_CFC_ (* Continuous Function Chart, elements in execution order *)
#0 OR(SCHU_P2_2_UE3_T_RESET, SCHU_P2_2_SB)
#1 SEL(UE3_T_FILTER_ON, T#0ms, T#2s)
#2 fb_UE3_T:ISTOK_ANALOGVH(enable: TRUE, rawValue: SCHU_P2_2_UE3_AI1, reset: #0, enableLimitCtrl: TRUE, ctrlVoltage: NOT UE3_T_CVOLT, changeValueWithoutPower: TRUE, highRange: UE_T_HIGHRANGE, lowRange: UE_T_LOWRANGE, highLimit: SCHU_P2_2_UE_T_HIGHLIMIT, lowLimit: SCHU_P2_2_UE_T_LOWLIMIT, filterTime: #1, offset: ofset, delayEnable: TE_DELAY)
#3 SCHU_P2_2_UE3_T_VN <= #2.presentValue
#4 SCHU_P2_2_UE3_T_DOST <= #2.reliability
#5 SUB(SCHU_P2_2_UE3_T_UST, 0.6)
#6 fb_UE3_m_UST:ISTOK_LT(dost: #2.reliability, x: #2.presentValue, ust: #5, shkal: -, gist: 0.5)
#7 SCHU_P2_2_UE3_TE_M_UST <= #6.Xm
#8 SCHU_P2_2_UE3_TE_B_UST <= #6.XmN
_END_CFC_
(* the same logic as Structured Text *)
fb_UE3_T(enable := TRUE, rawValue := SCHU_P2_2_UE3_AI1, reset := SCHU_P2_2_UE3_T_RESET OR SCHU_P2_2_SB, enableLimitCtrl := TRUE, ctrlVoltage := NOT UE3_T_CVOLT, changeValueWithoutPower := TRUE, highRange := UE_T_HIGHRANGE, lowRange := UE_T_LOWRANGE, highLimit := SCHU_P2_2_UE_T_HIGHLIMIT, lowLimit := SCHU_P2_2_UE_T_LOWLIMIT, filterTime := SEL(UE3_T_FILTER_ON, T#0ms, T#2s), offset := ofset, delayEnable := TE_DELAY);
SCHU_P2_2_UE3_T_VN := fb_UE3_T.presentValue;
SCHU_P2_2_UE3_T_DOST := fb_UE3_T.reliability;
fb_UE3_m_UST(dost := fb_UE3_T.reliability, x := fb_UE3_T.presentValue, ust := SCHU_P2_2_UE3_T_UST - 0.6, gist := 0.5);
SCHU_P2_2_UE3_TE_M_UST := fb_UE3_m_UST.Xm;
SCHU_P2_2_UE3_TE_B_UST := fb_UE3_m_UST.XmN;
END_PROGRAM

(* POU Input/AI/UE3_VL, CFC *)
PROGRAM UE3_VL
VAR
	fb_UE3_VL: ISTOK_ANALOGVH;
	ofset: REAL;
	fb_SCHU_P2_2_UE3_VL_B_UST: ISTOK_GT;
END_VAR
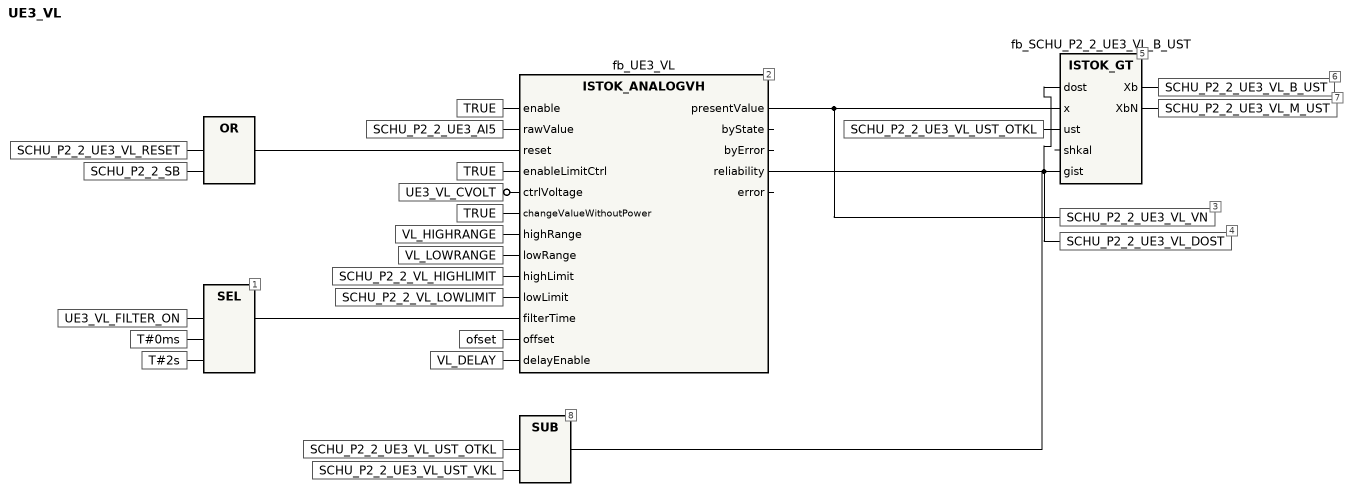
_CFC_ (* Continuous Function Chart, elements in execution order *)
#0 OR(SCHU_P2_2_UE3_VL_RESET, SCHU_P2_2_SB)
#1 SEL(UE3_VL_FILTER_ON, T#0ms, T#2s)
#2 fb_UE3_VL:ISTOK_ANALOGVH(enable: TRUE, rawValue: SCHU_P2_2_UE3_AI5, reset: #0, enableLimitCtrl: TRUE, ctrlVoltage: NOT UE3_VL_CVOLT, changeValueWithoutPower: TRUE, highRange: VL_HIGHRANGE, lowRange: VL_LOWRANGE, highLimit: SCHU_P2_2_VL_HIGHLIMIT, lowLimit: SCHU_P2_2_VL_LOWLIMIT, filterTime: #1, offset: ofset, delayEnable: VL_DELAY)
#3 SCHU_P2_2_UE3_VL_VN <= #2.presentValue
#4 SCHU_P2_2_UE3_VL_DOST <= #2.reliability
#5 fb_SCHU_P2_2_UE3_VL_B_UST:ISTOK_GT(dost: #2.reliability, x: #2.presentValue, ust: SCHU_P2_2_UE3_VL_UST_OTKL, shkal: -, gist: #8)
#6 SCHU_P2_2_UE3_VL_B_UST <= #5.Xb
#7 SCHU_P2_2_UE3_VL_M_UST <= #5.XbN
#8 SUB(SCHU_P2_2_UE3_VL_UST_OTKL, SCHU_P2_2_UE3_VL_UST_VKL)
_END_CFC_
END_PROGRAM

(* POU Input/AI/YA2_POS, CFC *)
PROGRAM YA2_POS
VAR
	ofset: REAL;
	fb_YA2: ISTOK_ANALOGVH;
	Lt_otkr_zakr: ISTOK_LT;
	gt_otkr_otr: ISTOK_GT;
	fb_YA2bUST_VKL_STER_REG: ISTOK_GT;
	fb_YA2mOTKL_STER_REG: ISTOK_LT;
END_VAR
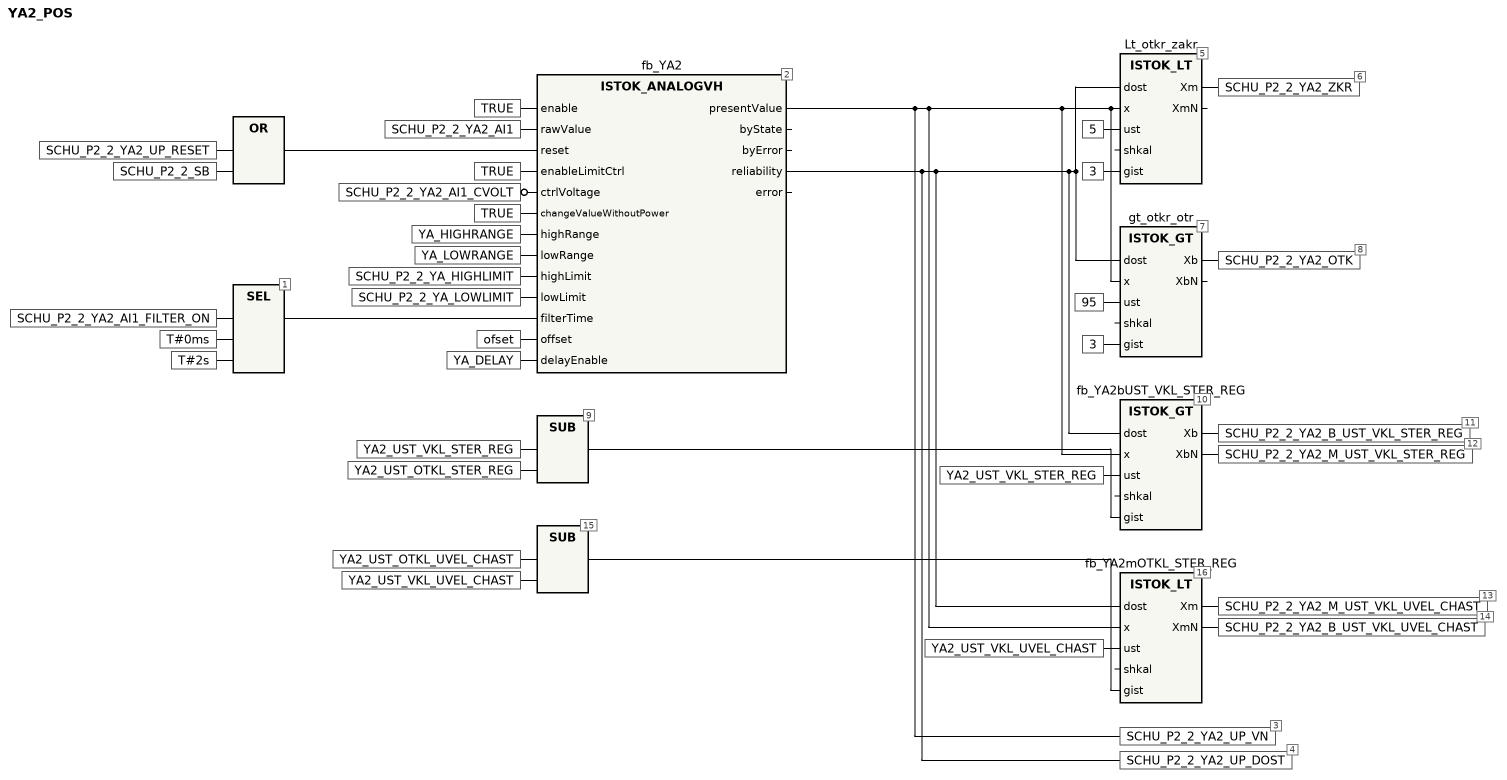
